// Mitsubishi GX Works2 project: program   PLC: Q03UDE

PROGRAM MAIN
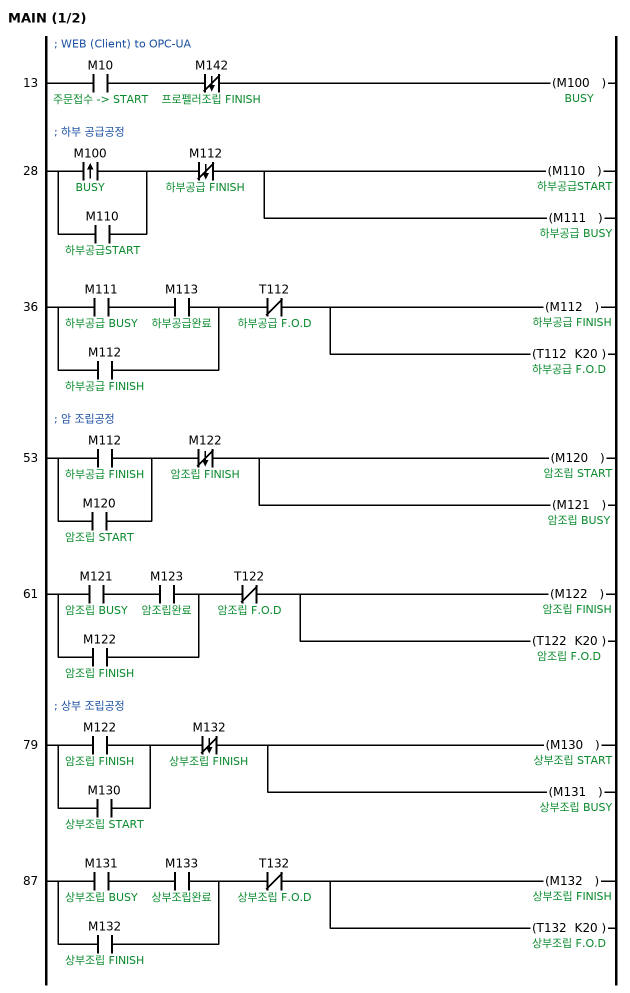
; WEB (Client) to OPC-UA
13    LD      M10  ; 주문접수 -> START
      ANDFI   M142  ; 프로펠러조립 FINISH
      OUT     M100  ; BUSY
; 하부 공급공정
28    LDP     M100  ; BUSY
      OR      M110  ; 하부공급START
      ANDFI   M112  ; 하부공급 FINISH
      OUT     M110  ; 하부공급START
      OUT     M111  ; 하부공급 BUSY
36    LD      M111  ; 하부공급 BUSY
      AND     M113  ; 하부공급완료
      OR      M112  ; 하부공급 FINISH
      ANI     T112  ; 하부공급 F.O.D
      OUT     M112  ; 하부공급 FINISH
      OUT     T112 K20  ; 하부공급 F.O.D
; 암 조립공정
53    LD      M112  ; 하부공급 FINISH
      OR      M120  ; 암조립 START
      ANDFI   M122  ; 암조립 FINISH
      OUT     M120  ; 암조립 START
      OUT     M121  ; 암조립 BUSY
61    LD      M121  ; 암조립 BUSY
      AND     M123  ; 암조립완료
      OR      M122  ; 암조립 FINISH
      ANI     T122  ; 암조립 F.O.D
      OUT     M122  ; 암조립 FINISH
      OUT     T122 K20  ; 암조립 F.O.D
; 상부 조립공정
79    LD      M122  ; 암조립 FINISH
      OR      M130  ; 상부조립 START
      ANDFI   M132  ; 상부조립 FINISH
      OUT     M130  ; 상부조립 START
      OUT     M131  ; 상부조립 BUSY
87    LD      M131  ; 상부조립 BUSY
      AND     M133  ; 상부조립완료
      OR      M132  ; 상부조립 FINISH
      ANI     T132  ; 상부조립 F.O.D
      OUT     M132  ; 상부조립 FINISH
      OUT     T132 K20  ; 상부조립 F.O.D
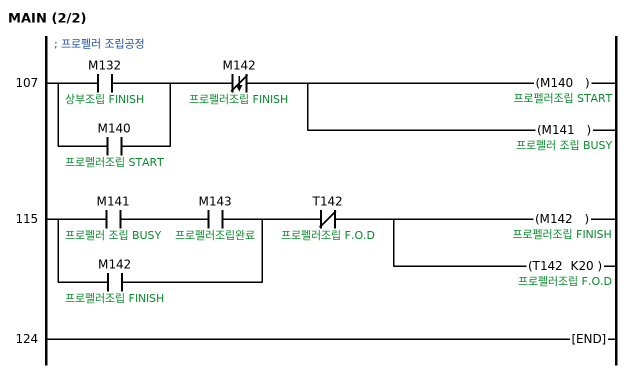
; 프로펠러 조립공정
107   LD      M132  ; 상부조립 FINISH
      OR      M140  ; 프로펠러조립 START
      ANDFI   M142  ; 프로펠러조립 FINISH
      OUT     M140  ; 프로펠러조립 START
      OUT     M141  ; 프로펠러 조립 BUSY
115   LD      M141  ; 프로펠러 조립 BUSY
      AND     M143  ; 프로펠러조립완료
      OR      M142  ; 프로펠러조립 FINISH
      ANI     T142  ; 프로펠러조립 F.O.D
      OUT     M142  ; 프로펠러조립 FINISH
      OUT     T142 K20  ; 프로펠러조립 F.O.D
124   END
END_PROGRAM

// device comments not shown above
T110  ; 하부공급 5초
T120  ; 암조립 20초
T130  ; 상부조립 5초
T140  ; 프로펠러 조립 15초
